(* Logix 5000 project; controller WP_Ottawa_Data_Concentrator_1 vendor 1 type 14 code 167 rev 32.14; software revision 32.04; part 5 of 5 *)
(* tags used below, declared in another part *)
   Array_Track : DINT;
   Local_Bool : BOOL[32];
   Local_DATETIME : DINT[10];
   Local_Timer : TIMER[5];
   ONS : BOOL[32];
   OPCFaultDateTime : STRING[10];
   str_DateTimeStamp : STRING[10];
   DC1_OPCFault : BOOL;
   DC1_OPCWatchDog : BOOL;
(* MainProgram, continued *)

ROUTINE MainRoutine   (* ladder *)
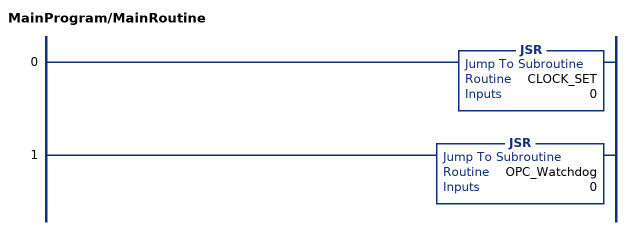
   0: JSR(CLOCK_SET,0);
   1: JSR(OPC_Watchdog,0);
END_ROUTINE

ROUTINE OPC_Watchdog   (* ladder *)
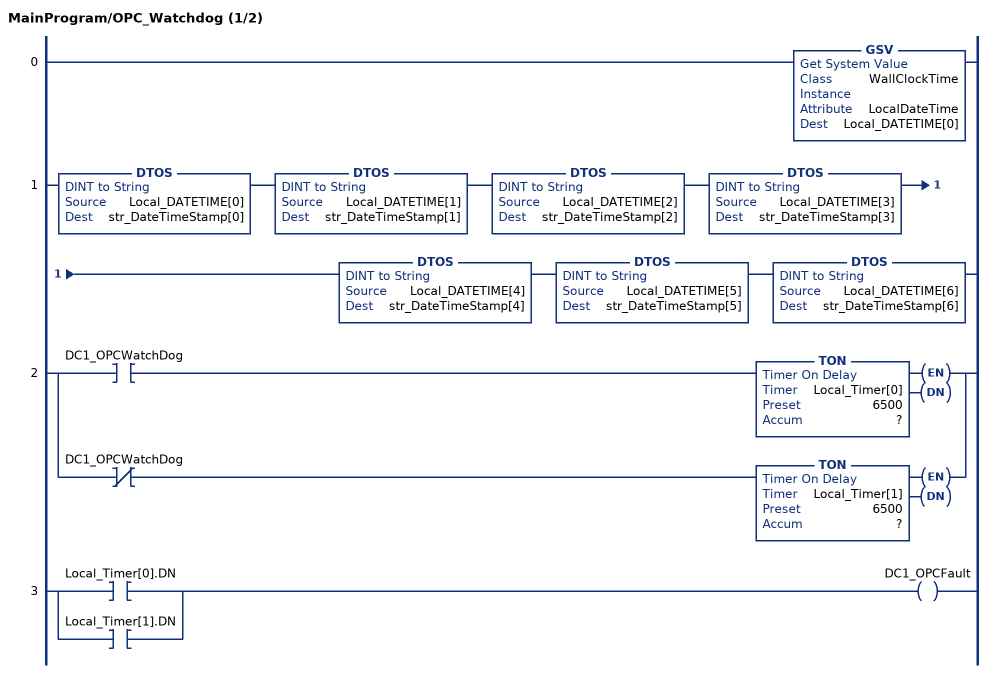
   0: GSV(WallClockTime,,LocalDateTime,Local_DATETIME[0]);
   1: DTOS(Local_DATETIME[0],str_DateTimeStamp[0])DTOS(Local_DATETIME[1],str_DateTimeStamp[1])DTOS(Local_DATETIME[2],str_DateTimeStamp[2])DTOS(Local_DATETIME[3],str_DateTimeStamp[3])DTOS(Local_DATETIME[4],str_DateTimeStamp[4])DTOS(Local_DATETIME[5],str_DateTimeStamp[5])DTOS(Local_DATETIME[6],str_DateTimeStamp[6]);
   2: [XIC(DC1_OPCWatchDog) TON(Local_Timer[0],?,?) ,XIO(DC1_OPCWatchDog) TON(Local_Timer[1],?,?) ];
   3: [XIC(Local_Timer[0].DN) ,XIC(Local_Timer[1].DN) ]OTE(DC1_OPCFault);
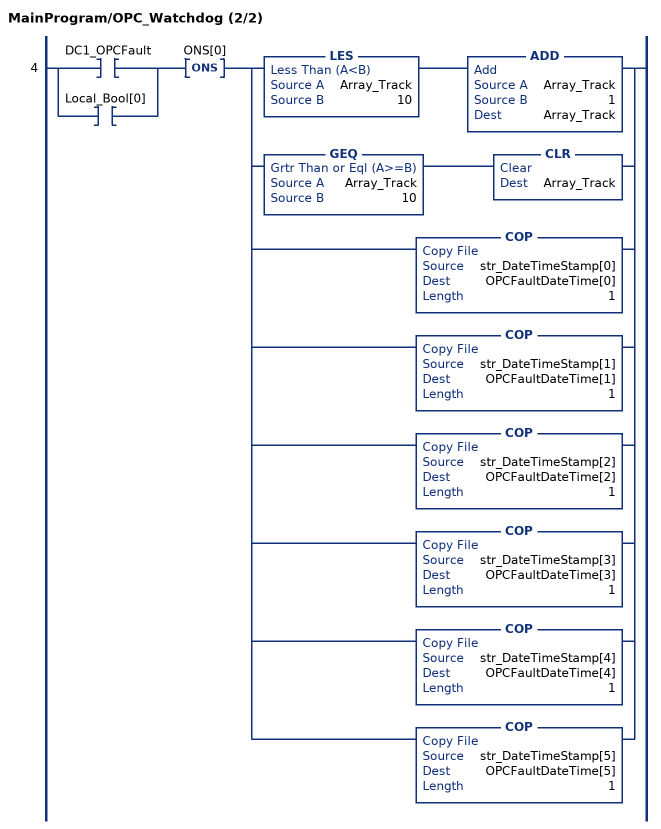
   4: [XIC(DC1_OPCFault) ,XIC(Local_Bool[0]) ]ONS(ONS[0])[LES(Array_Track,10) ADD(Array_Track,1,Array_Track) ,GEQ(Array_Track,10) CLR(Array_Track) ,COP(str_DateTimeStamp[0],OPCFaultDateTime[0],1) ,COP(str_DateTimeStamp[1],OPCFaultDateTime[1],1) ,COP(str_DateTimeStamp[2],OPCFaultDateTime[2],1) ,COP(str_DateTimeStamp[3],OPCFaultDateTime[3],1) ,COP(str_DateTimeStamp[4],OPCFaultDateTime[4],1) ,COP(str_DateTimeStamp[5],OPCFaultDateTime[5],1) ];
END_ROUTINE
END_PROGRAM
